// TIA Portal V20 export
DATA_BLOCK "ControlNodes"   // DB174
// stored: MemoryReserve 100, Namespace Unit1.Em4
   VAR
      em : "LAF_typeEmControlNode";
      emstate { S7_SetPoint := 'True'} : "LUC_typeStates";
      cm : "Unit1.Em4.typeCmControlNode";
      citiMap : Struct
         PMC : "LER_PMC_Input_Data";
         FlexNet { S7_SetPoint := 'True'} : "LER_FlexNet_Data";
      END_STRUCT;
      sideTapeLoading : "Unit1.Em4.typeSequenceControlNode_sideTapeLoading";
      sideTapeAttachment : "Unit1.Em4.typeSequenceControlNode_sideTapeAttachment";
      sideTapeFixStage : "Unit1.Em4.typeSequenceControlNode_sideTapeFixStage";
      SpecialFunctionMode : Struct
         DryRun : Struct
            JRdetectPV : Array[0..15] of Bool;
         END_STRUCT;
      END_STRUCT;
      cmSideTapeSafetyPin : "LBC_typeDigitalSignalControlNode";
      cmSideTapeJRDetect : "LBC_typeDigitalSignalControlNode";
      cmSideTapeDiameter : "LBC_typeDigitalSignalControlNode";
      cmSideTapeFixStageAxisX : "LBC_typeAxis64PosControlNode";
      cmSideTapeFixStageAxisC : "LBC_typeAxis64PosControlNode";
      cmSideTapeAttachmentAxisX : "LBC_typeAxis64PosControlNode";
      cmSideTapeAttachmentAxisY : "LBC_typeAxis64PosControlNode";
      cmSideTapeLoadingDownUp : "LBC_typeTwoWayActuatorControlNode";
      cmSideTapeLoadingClampOpenClose : "LBC_typeTwoWayActuatorControlNode";
      cmSideTapeCutterBwdFwd : "LBC_typeTwoWayActuatorControlNode";
      cmSideTapeCutterClampBwdFwd : "LBC_typeTwoWayActuatorControlNode";
      cmSideTapeTensionBwdFwd : "LBC_typeTwoWayActuatorControlNode";
      cmSideTapeAttachmentLeftBwdFwd : "LBC_typeTwoWayActuatorControlNode";
      cmSideTapeAttachmentRightBwdFwd : "LBC_typeTwoWayActuatorControlNode";
      cmSideTapeAttachmentBtmBwdFwd : "LBC_typeTwoWayActuatorControlNode";
      cmSideTapeFixStageClampOpenClose : "LBC_typeTwoWayActuatorControlNode";
      cmSideTapeAttachment1TopVaccumOffOn : "LBC_typeTwoWayActuatorControlNode";
      cmSideTapeAttachment1BtmVaccumOffOn : "LBC_typeTwoWayActuatorControlNode";
      cmSideTapeAttachment2TopVaccumOffOn : "LBC_typeTwoWayActuatorControlNode";
      cmSideTapeAttachment2BtmVaccumOffOn : "LBC_typeTwoWayActuatorControlNode";
      cmQrHandyReader : "LER_typeDM8700ControlNode";
   END_VAR
BEGIN
   em.status.enabled := true;
END_DATA_BLOCK
